TYPE ST_CoeEntry_REAL EXTENDS ST_CoeEntry :
STRUCT
	Value	: REAL;
END_STRUCT
END_TYPE

(* stored: Version 1.1.0.1, ProductVersion 3.1.4024.13
   DUT ST_CoeEntry_REAL: Id {4d515ae5-5e80-06b0-0413-aaec91028fde} *)
